# EPICS autosave request: i404App/Db/I404.req
#FILE... I404.req

$(DEVICE):INITMODE
$(DEVICE):RANGE_
$(DEVICE):SCNERR.SCAN
$(DEVICE):FREQ
$(DEVICE):GETCS.SCAN
$(DEVICE):Resolution
$(DEVICE):SuppressFreq
